// LS Electric XG5000 project: 터치연습11
// PLC LSPLC

PROGRAM NewProgram (task: 스캔 프로그램)

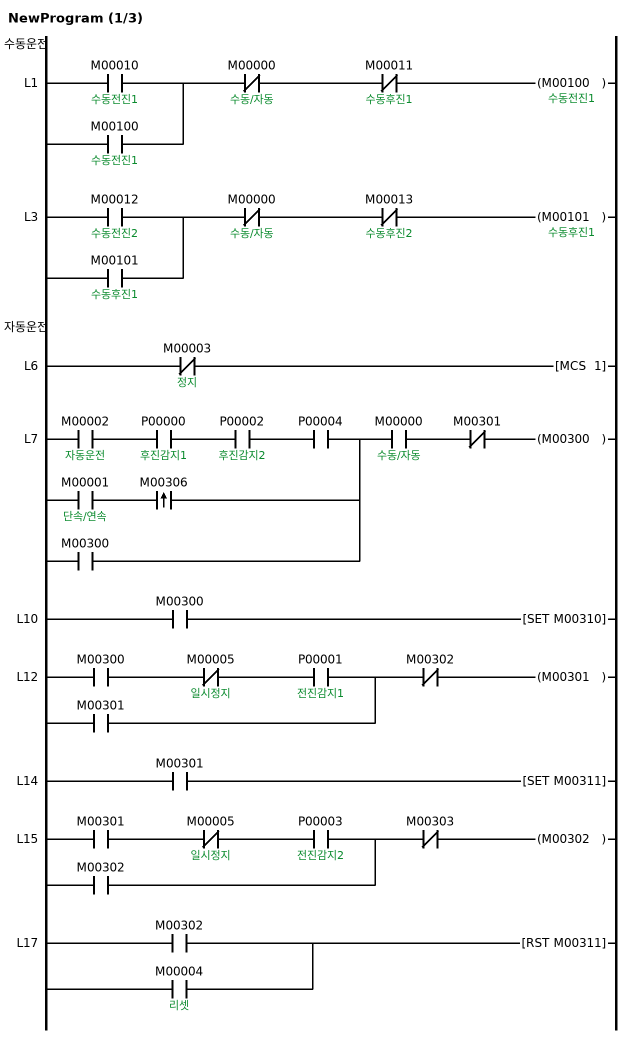
수동운전:
; L1
LOAD      M00010	// 수동전진1
OR        M00100	// 수동전진1
AND NOT   M00000	// 수동/자동
AND NOT   M00011	// 수동후진1
OUT       M00100	// 수동전진1
; L3
LOAD      M00012	// 수동전진2
OR        M00101	// 수동후진1
AND NOT   M00000	// 수동/자동
AND NOT   M00013	// 수동후진2
OUT       M00101	// 수동후진1
자동운전:
; L6
LOAD NOT  M00003	// 정지
MCS       1
; L7
LOAD      M00002	// 자동운전
AND       P00000	// 후진감지1
AND       P00002	// 후진감지2
AND       P00004
LOAD      M00001	// 단속/연속
ANDP      M00306
OR LOAD
OR        M00300
AND       M00000	// 수동/자동
AND NOT   M00301
OUT       M00300
; L10
LOAD      M00300
SET       M00310
; L12
LOAD      M00300
AND NOT   M00005	// 일시정지
AND       P00001	// 전진감지1
OR        M00301
AND NOT   M00302
OUT       M00301
; L14
LOAD      M00301
SET       M00311
; L15
LOAD      M00301
AND NOT   M00005	// 일시정지
AND       P00003	// 전진감지2
OR        M00302
AND NOT   M00303
OUT       M00302
; L17
LOAD      M00302
OR        M00004	// 리셋
RST       M00311

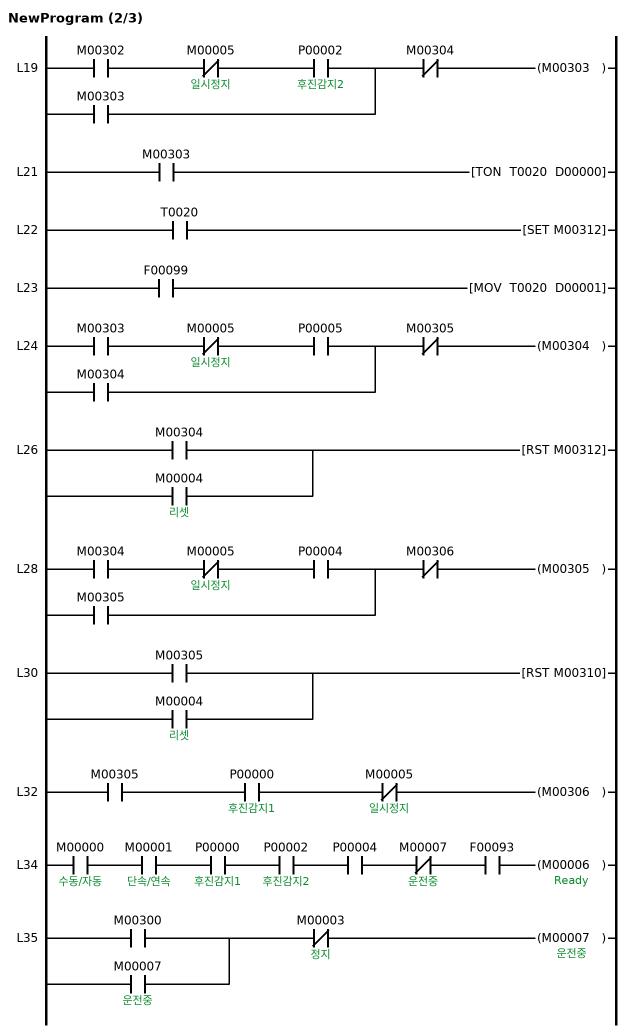
; L19
LOAD      M00302
AND NOT   M00005	// 일시정지
AND       P00002	// 후진감지2
OR        M00303
AND NOT   M00304
OUT       M00303
; L21
LOAD      M00303
TON       T0020 D00000
; L22
LOAD      T0020
SET       M00312
; L23
LOAD      F00099
MOV       T0020 D00001
; L24
LOAD      M00303
AND NOT   M00005	// 일시정지
AND       P00005
OR        M00304
AND NOT   M00305
OUT       M00304
; L26
LOAD      M00304
OR        M00004	// 리셋
RST       M00312
; L28
LOAD      M00304
AND NOT   M00005	// 일시정지
AND       P00004
OR        M00305
AND NOT   M00306
OUT       M00305
; L30
LOAD      M00305
OR        M00004	// 리셋
RST       M00310
; L32
LOAD      M00305
AND       P00000	// 후진감지1
AND NOT   M00005	// 일시정지
OUT       M00306
; L34
LOAD      M00000	// 수동/자동
AND       M00001	// 단속/연속
AND       P00000	// 후진감지1
AND       P00002	// 후진감지2
AND       P00004
AND NOT   M00007	// 운전중
AND       F00093
OUT       M00006	// Ready
; L35
LOAD      M00300
OR        M00007	// 운전중
AND NOT   M00003	// 정지
OUT       M00007	// 운전중

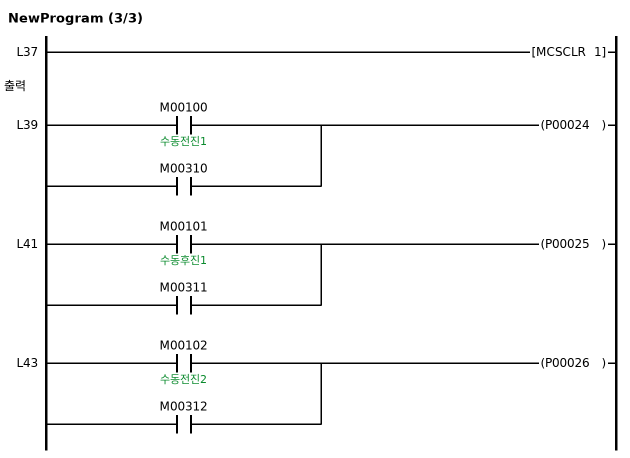
; L37
MCSCLR    1
출력:
; L39
LOAD      M00100	// 수동전진1
OR        M00310
OUT       P00024
; L41
LOAD      M00101	// 수동후진1
OR        M00311
OUT       P00025
; L43
LOAD      M00102	// 수동전진2
OR        M00312
OUT       P00026

VARIABLES AND COMMENTS (devices not used above)
P00020	BIT	전진1
M00103	BIT	수동후진2
P00021	BIT	후진1
P00022	BIT	전진2
P00023	BIT	후진2
M00200	BIT	전진1
M00201	BIT	전진2
M00202	BIT	후진1
M00203	BIT	후진2
M00204	BIT	2후진 완료